FUNCTION_BLOCK FB_Normalize_1
// INT: [-32768, 32767]	
// LREAL: Long Real decimal number

// Constant variables
VAR CONSTANT
	MaxBitValue : LREAL := 32767.0;
END_VAR

// Input variables
VAR_INPUT
	nRawInput : INT;
	fMaxValue : LREAL;
END_VAR

// Output variables
VAR_OUTPUT
	fNormalizedInput : LREAL;
END_VAR

fNormalizedInput := (fMaxValue	* INT_TO_LREAL(nRawInput)) / MaxBitValue;
// Value/Max-value = Raw_value/Max-raw_value. Uses this definition to calculate value for normalized data.
// Int_to_Lreal makes an integer into a long real decimal number
// 16 bit = [-32767, 32767], max value: 32 767

fNormalizedInput := LIMIT(0, fNormalizedInput, fMaxValue); // Limit(min, test-value, max)
// Safety function. Lowest value = 0, highest = f_MaxValue

END_FUNCTION_BLOCK

(* stored: Version 1.1.0.1
   POU FB_Normalize_1: Id {a78fb5e3-d685-4d3d-9971-5c4c25d20393}, SpecialFunc None *)
